(* PLC project OOP_Curso, Beckhoff Automation GmbH TwinCAT PLC Control 3.5.13.21 *)
(* stored: creationDateTime 2023-07-27T12:50:36.7292719, modificationDateTime 2023-07-27T12:50:36.7361023 *)

TYPE ST_Empleado :
STRUCT
	Nombre 				: STRING;
    Apellido 			: STRING;
    CorreoElectronico 	: STRING;
END_STRUCT
END_TYPE

TYPE ST_Horario :
STRUCT
	HoraEntrada : DATE_AND_TIME;
    HoraSalida : DATE_AND_TIME;
END_STRUCT
END_TYPE

TYPE ST_RegistroDeTiempoEmpleado :
STRUCT
	stEmpleado : ST_Empleado; // Datos de la función Empleado
    stHorario  : ST_Horario;
END_STRUCT
END_TYPE

FUNCTION_BLOCK FB_Empleado
VAR_INPUT
	stEmpleado :ST_Empleado;
END_VAR
VAR_OUTPUT
END_VAR
VAR
	_Empleado : ST_Empleado;
END_VAR

            
          

METHOD FB_init : BOOL
VAR_INPUT
	bInitRetains : BOOL; // if TRUE, the retain variables are initialized (warm start / cold start)
	bInCopyCode : BOOL;  // if TRUE, the instance afterwards gets moved into the copy code (online change)
	Empleado : ST_Empleado;
END_VAR
                  _Empleado := Empleado;
                
END_METHOD

PROPERTY Apellido : STRING
GET
VAR
END_VAR
                    Apellido := _Empleado.Apellido;
                  
END_GET
SET
VAR
END_VAR
                    _Empleado.Apellido := Apellido;
                  
END_SET
END_PROPERTY

PROPERTY CorreoElectronico : STRING
GET
VAR
END_VAR
                    CorreoElectronico := _Empleado.CorreoElectronico;
                  
END_GET
SET
VAR
END_VAR
                     _Empleado.CorreoElectronico := CorreoElectronico;
                  
END_SET
END_PROPERTY

PROPERTY Nombre : STRING
GET
VAR
END_VAR
                    Nombre := _Empleado.Nombre;
                  
END_GET
SET
VAR
END_VAR
                    _Empleado.Nombre := Nombre;
                  
END_SET
END_PROPERTY
END_FUNCTION_BLOCK

FUNCTION_BLOCK FB_RegistroDeTiempo
VAR_INPUT
	stEmpleado : ST_Empleado; // instancia de la función Empleado
    stHorario  : ST_Horario;
END_VAR
VAR_OUTPUT
END_VAR
VAR
	_RegistroDeTiempo : ST_RegistroDeTiempoEmpleado;
END_VAR

            
          

METHOD FB_init : BOOL
VAR_INPUT
	bInitRetains : BOOL; // if TRUE, the retain variables are initialized (warm start / cold start)
	bInCopyCode : BOOL;  // if TRUE, the instance afterwards gets moved into the copy code (online change)
	RegistroDeTiempo : ST_RegistroDeTiempoEmpleado;
END_VAR
                  _RegistroDeTiempo := RegistroDeTiempo;
                
END_METHOD

PROPERTY Empleado : ST_Empleado;
GET
VAR
END_VAR
                    
                  
END_GET
SET
VAR
END_VAR
                    
                  
END_SET
END_PROPERTY

PROPERTY HoraEntrada : DATE_AND_TIME
GET
VAR
END_VAR
                    
                  
END_GET
SET
VAR
END_VAR
                    
                  
END_SET
END_PROPERTY

PROPERTY HoraSalida : DATE_AND_TIME
GET
VAR
END_VAR
                    
                  
END_GET
SET
VAR
END_VAR
                    
                  
END_SET
END_PROPERTY
END_FUNCTION_BLOCK

PROGRAM _24_SOLID_SRP
VAR
	stRaul 						: ST_Empleado := (Nombre:= 'Raul', Apellido:= 'Gonzalez', CorreoElectronico:= 'micorreo@correo.com');
	Empleado_1 					: FB_Empleado(stRaul);
	
	stHorario_Raul 				: ST_Horario := (HoraEntrada := DT#2023-1-1-8:0:0, HoraSalida := DT#2023-1-1-17:0:0);
	stRegistroDeTiempoEmpleado 	: ST_RegistroDeTiempoEmpleado := (stEmpleado:= stRaul, stHorario:= stHorario_Raul);
	RegistroDeTiempoEmpleado_1 : FB_RegistroDeTiempo(stRegistroDeTiempoEmpleado);
	
	
END_VAR

            
          
END_PROGRAM
